Staubli VAL3: strfill.pgx

public program strfill(string pStrIn (dimensions=1), num pLenStrOut (dimensions=1), string& pStrOut[] (dimensions=1))
  local string lEmpty
  local num lLen
begin
  //---------------------------------
  //  F I L L   O N E   S T R I N G
  //---------------------------------
  // To fill the string with space
  // character
  //
  // look for asian message
  if getDisplayLen(pStrIn)<pLenStrOut
    // insert some space
    lEmpty="                                        "
    pStrOut=pStrIn
    lLen=(pLenStrOut-getDisplayLen(pStrIn))
    call midPos(lEmpty,lLen,0,pStrIn)
    pStrOut=pStrOut+pStrIn
  else
    if getDisplayLen(pStrIn)>pLenStrOut
      // divide the string
      call midPos(pStrIn,pLenStrOut,0,pStrOut)
    else
      // they are the same
      pStrOut=pStrIn
    endIf
  endIf
end
